{attribute 'linkalways'} 
{attribute 'no_explicit_call' := 'This FB is a CLASS and must be accessed using methods or properties'}
{attribute 'enable_dynamic_creation'}
FUNCTION_BLOCK FINAL NOT_WORD EXTENDS Node
VAR
	in : _WORD(0);
	out : _WORD(0);
END_VAR

METHOD PUBLIC Clone : I_Node
VAR
	pNode : POINTER TO NOT_WORD;
END_VAR
pNode := __NEW(NOT_WORD);
Clone := pNode^;
END_METHOD

METHOD FB_init : BOOL
VAR_INPUT
	bInitRetains : BOOL; // if TRUE, the retain variables are initialized (warm start / cold start)
	bInCopyCode : BOOL;  // if TRUE, the instance afterwards gets moved into the copy code (online change)
END_VAR
AddInput('in',THIS^.in);
AddOutput('out', THIS^.out);
END_METHOD

METHOD PROTECTED OnExecute
VAR
END_VAR
out.Value := NOT in.Value;
END_METHOD

END_FUNCTION_BLOCK

(* stored: Version 1.1.0.1, ProductVersion 3.1.4024.15
   POU NOT_WORD: Id {83fe150a-acf8-4792-a612-df27af6b021c}, SpecialFunc None
   Folder Constructor: Id {176b83aa-c7c2-4755-9723-e1aab581ce75}
   Method Clone: Id {801845c3-5e02-4401-ad76-9ade3e47f1e3}
   Method FB_init: Id {22aaa58c-8990-49cb-867d-4f4bf8e7c8e5}
   Method OnExecute: Id {50a7c6e0-1a1c-4e58-abdd-e17b3c3f559c} *)
